PROGRAM BH0HPL_LineBackground
VAR
END_VAR

MAIN.stLine_BH0GPL.fbLine(stLine:=MAIN.stLine_BH0GPL);
MAIN.stLine_BH0GPL.stStation_BH0GPL01.fbStation(
				stLine:=MAIN.stLine_BH0GPL,
				stStation:=MAIN.stLine_BH0GPL.stStation_BH0GPL01);

END_PROGRAM

(* stored: Version 1.1.0.1, ProductVersion 3.1.4024.15
   POU BH0HPL_LineBackground: Id {dd96c757-0e3d-42d7-8224-5399c89c3c3f}, SpecialFunc None *)
